Fanuc KAREL source: kt00046.KL

-- PROVISIONAL review KL for V1013-1; original PC SHA256 13c47fea89820632a8a8ae8674500b69ce2f6cd4acb4560b1096c6b68671f519
-- Incomplete behavior may be omitted. Consult companion uncertainty JSON. Do not deploy.
PROGRAM KT00046
%NOLOCKGROUP
VAR
  R1 : REAL
  OUT : REAL
-- UNRESOLVED_DECL Y2 type=002018
BEGIN
  -- UNRESOLVED_PC offsets 5-16; opcodes 2E,23
  -- UNRESOLVED_PC offsets 21-35; opcodes 2E,22,9D,33,B2
  -- UNRESOLVED_PC offsets 40-63; opcodes 21,22,9D,33,B1,64,6A,23
  -- UNRESOLVED_PC offsets 68-72; opcodes 7F
END KT00046
